{attribute addProperty BoxType "EK1100-0000-0018"}
{attribute addProperty Id "Beckhoff_EJ9xxxEK1122Beckhoff_EJ9xxxEK1122_DB893B98162A_0001_EJ9001_0000_0016EJ9001_179A0949162A_0002_EJ9505_0000_0016EJ9505_A1085FEB486A_0003_EJ9576_0000_0018EJ9576_37EDA20522428A_0004_EJ9576_0000_0019EJ9576_A45E449923229A_0005_EJ9576_0000_0020EJ9576_57CA9E3622428A_0006_EJ9576_0000_0022EJ9576_B5DF83EF23229"}
{attribute addProperty CRC "361647231"}
{attribute addProperty SizeInBites "992"}
{attribute addProperty SizeInBytes "124"}
TYPE Beckhoff_EJ9xxx_158E4C7F EXTENDS EK1100_179A0949 :
STRUCT
	{attribute addProperty Name "Beckhoff_EJ9xxxEK1122"}
	Beckhoff_EJ9xxxEK1122 : Beckhoff_EJ9xxxEK1122_DB893B98;
	{attribute addProperty Name "A_0001_EJ9001_0000_0016"}
	A_0001_EJ9001_0000_0016 : EJ9001_179A0949;
	{attribute addProperty Name "A_0002_EJ9505_0000_0016"}
	A_0002_EJ9505_0000_0016 : EJ9505_A1085FEB;
	{attribute addProperty Name "A_0003_EJ9576_0000_0018"}
	A_0003_EJ9576_0000_0018 : EJ9576_37EDA205;
	{attribute addProperty Name "A_0004_EJ9576_0000_0019"}
	A_0004_EJ9576_0000_0019 : EJ9576_A45E4499;
	{attribute addProperty Name "A_0005_EJ9576_0000_0020"}
	A_0005_EJ9576_0000_0020 : EJ9576_57CA9E36;
	{attribute addProperty Name "A_0006_EJ9576_0000_0022"}
	A_0006_EJ9576_0000_0022 : EJ9576_B5DF83EF;
END_STRUCT
END_TYPE

(* stored: Version 1.2.0.0, ProductVersion 3.1.4024.9
   DUT Beckhoff_EJ9xxx_158E4C7F: Id {807b692b-5e91-4444-84de-aa3bdc256df9} *)
